// TwinCAT 3 PLC project LatchSR
// ProgramVersion: 3.1.4023.0
// libraries:
//   Tc2_Standard, * (Beckhoff Automation GmbH)
//   Tc2_System, * (Beckhoff Automation GmbH)
//   Tc3_Module, * (Beckhoff Automation GmbH)
// project tree:
//   GVLs/ GVL.TcGVL
//   / PlcTask.TcTTO
//   POUs/ MAIN.TcPOU
// real-time tasks:
//   TASK PlcTask: cycle T#10ms, priority 20, ADS port 350
// I/O:
//   DEVICE Dispositivo 1 (EtherCAT), AmsNetId 5.71.198.244.2.1
//     Terminale 1 (EK1200) [EK1200-5000 EtherCAT Power supply (2A E-Bus)]
//       Terminale 2 (EL1008) [EL1008 8Ch. Dig. Input 24V, 3ms]
//       Terminale 3 (EL2008) [EL2008 8Ch. Dig. Output 24V, 0.5A]
//       Terminale 4 (EL3064) [EL3064 4Ch. Ana. Input 0-10V]
//       Terminale 5 (EL4002) [EL4002 2Ch. Ana. Output 0-10V, 12bit]
//       Terminale 6 (EL7031) [EL7031 1Ch. Stepper motor output stage (24V, 1.5A)]
//       Terminale 7 (EL3202) [EL3202 2Ch. Ana. Input PT100 (RTD)]
//       Terminale 8 (EL4022) [EL4022 2Ch. Ana. Output 4-20mA, 12bit]
//       Terminale 9 (EL9011) [EL9011 End Terminal]
// variable links:
//   LatchSR/LatchSR Instance <-> Device 1 (EtherCAT)/Term 1 (EK1200)/Term 2 (EL1008)
//     PlcTask Inputs/GVL.bDigital_Inputs[1] <-> Channel 1/Input
//     PlcTask Inputs/GVL.bDigital_Inputs[2] <-> Channel 2/Input
//   LatchSR/LatchSR Instance <-> Device 1 (EtherCAT)/Term 1 (EK1200)/Term 3 (EL2008)
//     PlcTask Outputs/GVL.bDigital_Outputs[1] <-> Channel 1/Output

CONFIGURATION LatchSR
    RESOURCE PLC ON TwinCAT3
        TASK PlcTask(INTERVAL := T#10ms, PRIORITY := 20);
        PROGRAM MAIN WITH PlcTask : MAIN;
    END_RESOURCE
END_CONFIGURATION

// ---- GVLs/GVL.TcGVL
{attribute 'qualified_only'}
VAR_GLOBAL
	bDigital_Inputs AT %I* : ARRAY[1..8] OF BOOL;
	bDigital_Outputs AT %Q* : ARRAY[1..8] OF BOOL;
END_VAR

// ---- POUs/MAIN.TcPOU
PROGRAM MAIN
VAR
	fbSR : SR;
END_VAR

fbSR(SET1:= GVL.bDigital_Inputs[1], RESET:= GVL.bDigital_Inputs[2]);

GVL.bDigital_Outputs[1] := fbSR.Q1;
GVL.bDigital_Outputs[2] := fbSR.Q1;
GVL.bDigital_Outputs[3] := fbSR.Q1;
GVL.bDigital_Outputs[4] := fbSR.Q1;
GVL.bDigital_Outputs[5] := fbSR.Q1;
GVL.bDigital_Outputs[6] := fbSR.Q1;

END_PROGRAM
